(* Logix 5000 project; controller Battleship Emulate 5570 rev 32.11; software revision 32.00 *)

TASK MainTask (continuous, watchdog 500 ms) : MainProgram, Player_2, Player_1

MODULES
   Local : Emulate 5570 (ICP 2, rev 32.11)
END_MODULES

TYPE HMI_ScreenNames :
STRUCT
   LoadingScreen : STRING;
   BattleScreen : STRING;
END_STRUCT
END_TYPE

TYPE PlayerData :
STRUCT
   Ship : Ship[6];
   HMI : PlayerHMI;
   sName : STRING;
   nScore : INT;
   ShipSelectedFromFleet : SINT;
   sideShipSelected_ID : SINT;
   anySideShipSelected : BOOL;
   bShipsDeployed : BOOL;
   bTacticalScreenEnabled : BOOL;
   bBattleScreenEnabled : BOOL;
   bTurn : BOOL;
   bWinner : BOOL;
END_STRUCT
END_TYPE

TYPE PlayerHMI :
STRUCT
   sLoad_Or_Battle : STRING;   // The name of the screen that will load after player presses the Ready button
   bResetBoard_PB : BOOL;
   bRetrieveShip_PB : BOOL;
   bRetrieveShipPB_Vis : BOOL;
   bShipPiece_Orientation_PB : BOOL;
   bReady_PB : BOOL;   // Player Ready Signal from HMI
   bEnableStartPB : BOOL;   // Enable Start button on HMI
   bFight_PB : BOOL;
   bFightPB_Vis : BOOL;
   bWaitingForOpponent : BOOL;
END_STRUCT
END_TYPE

TYPE Ship :
STRUCT
   Position : INT[2];   // X-Y Ship Coordinates
   Pivot : INT[2];   // X-Y Pivot Coordinates
   nShipID : SINT;
   nShipLength : SINT;   // 5 = Carrier 4 = Battleship 3 = Cruiser 2 = Destroyer
   bIsHit : BOOL;
   bIsSunked : BOOL;
   bIsSelected : BOOL;
   bHideSidePiece : BOOL;
END_STRUCT
END_TYPE

TYPE Tile :
STRUCT
   IND : SINT;   // 0 = No ship 1 = Has ship 2 = Has ship and selected
   ShipID : SINT;
   hasShip : BOOL;
   squareSelected : BOOL;
END_STRUCT
END_TYPE

TYPE TileSelection :
STRUCT
   Coordinate : XYcoordinates;
   ShipId : DINT;
END_STRUCT
END_TYPE

TYPE top_scrn :
STRUCT
   notSelected : BOOL;
   selected : BOOL;
   hit : BOOL;
END_STRUCT
END_TYPE

TYPE XYcoordinates :
STRUCT
   row : SINT;
   column : SINT;
END_STRUCT
END_TYPE

ADD_ON_INSTRUCTION BattleTracker   (* revision 1.0 *)
VAR_IN_OUT
   TileSelected : TileSelection; {required}
   OtherPlayer_TS : Tile[11,11]; {required}
   BattleScreen : Tile[11,11]; {required}
   OtherPlayer : PlayerData; {required}
   ThisPlayer : PlayerData; {required}
END_VAR
VAR
   row : DINT; {access None}
   column : DINT; {access None}
END_VAR

ROUTINE Logic   (* structured text *)
   if OtherPlayer_TS[TileSelected.Coordinate.row, TileSelected.Coordinate.column].hasShip then
   	BattleScreen[TileSelected.Coordinate.row, TileSelected.Coordinate.column].IND := 4;
   	ThisPlayer.nScore := ThisPlayer.nScore + 1;
   else
   	BattleScreen[TileSelected.Coordinate.row, TileSelected.Coordinate.column].IND := 3;
   end_if;
   
   
   TileSelected.Coordinate.row := 0;
   TileSelected.Coordinate.column := 0;
   
   // Terminate player's turn
   ThisPlayer.bTurn := 0;
   OtherPlayer.bTurn := 1;
   
   
END_ROUTINE
END_ADD_ON_INSTRUCTION

ADD_ON_INSTRUCTION CommandShip   (* revision 1.0 *)
VAR_IN_OUT
   Player_Ship : Ship[5]; {required}
   Player_tacticalScreen : Tile[10,10]; {required}
END_VAR
VAR_INPUT
   verticalOrientation : BOOL; {required}
   NumberOfShips : DINT; {access Read Only, required}
END_VAR
VAR_IN_OUT
   shipSelected : SINT; {required}
END_VAR
VAR
   selectedSquare : XYcoordinates; {access None}
   x : DINT; {access None}
   row : DINT; {access None}
   column : DINT; {access None}
END_VAR

ROUTINE Logic   (* structured text *)
   // Initialize variables
   //shipSelected := -1;
   selectedSquare.row := -1;
   selectedSquare.column := -1;
   /*
   
   // Look for any side ship that was selected from the side pieces
   // shipSelected = the ship the was selected from the side pieces
   for x := 0 to NumberOfShips-1 by 1  do
   	//anySelected := 0;
   	if Player_Ship[x].isSelected then
   		shipSelected := x;
   		selectedSquare.row := -1;
   		selectedSquare.column := -1;
   	else
   		shipSelected := -1;
   		selectedSquare.row := -1;
   		selectedSquare.column := -1;
   	end_if;
   	/*
   	anySelected := ThisPlayer.Ship[x].isSelected OR anySelected;
   	if not anySelected then
   		shipSelected := -1;
   	end_if;
   
   
   end_for;
   
   */
   
   
   
   // If a ship piece was selected, enable search to look for the square that gets selected on the tactical screen
   // Store the XY coordinates of the selected square in selectedSquare.row and selectedSquare.column
   if shipSelected >= 0 then
   	for row := 0 to 9 by 1 do
   		for column := 0 to 9 by 1 do
   			if Player_tacticalScreen[row,column].squareSelected then
   				selectedSquare.row := row;
   				selectedSquare.column := column;
   				Player_tacticalScreen[row,column].squareSelected := 0;
   			end_if;
   		end_for;
   	end_for;
   end_if;
   
   
   /*
   // If a ship piece and a square were selected,
   // set the adjacent squares "hasShip" to 1 horizontally starting with the selected ship and moving to the right for as many squares as the ship's length
   if selectedSquare.row <> -1 AND selectedSquare.column <> -1 then
   
   	if verticalOrientation then		// Place ship in vertical orientation
   		for column := selectedSquare.column to selectedSquare.column + Player_Ship[x].shipLength -1 by 1 do
   			Player_tacticalScreen[selectedSquare.row,column].hasShip := 1;
   			Player_tacticalScreen[selectedSquare.row,column].hasShipType := shipSelected;
   			Player_tacticalScreen[selectedSquare.row,column].IND := 1;
   			Player_Ship[shipSelected].isSelected := 0;
   		end_for;
   
   
   	else	// Place ship in horizontal orientation
   		for row:= selectedSquare.row to selectedSquare.row + Player_Ship[x].shipLength -1 by 1 do
   			Player_tacticalScreen[row,selectedSquare.column].hasShip := 1;
   			Player_tacticalScreen[row,selectedSquare.column].hasShipType := shipSelected;
   			Player_tacticalScreen[row,selectedSquare.column].IND := 1;
   			Player_Ship[shipSelected].isSelected := 0;
   		end_for;
   	end_if;
   end_if;
   
   
   /*
   TODO
   
   add vertical/horizontal button and adjust how you lay the ship accordingly
   
   add retrieve button
   
   count down the ship pieces. disable piece once count reaches zero
   */
END_ROUTINE
END_ADD_ON_INSTRUCTION

ADD_ON_INSTRUCTION heartBeat   (* revision 1.0 *)
VAR_INPUT
   onTime : DINT; {required}
   offTime : DINT; {required}
END_VAR
VAR_OUTPUT
   Beat : BOOL; {access None, visible}
END_VAR
VAR
   T2 : TIMER; {access None}
   T1 : TIMER; {access None}
END_VAR

ROUTINE Logic   (* ladder *)
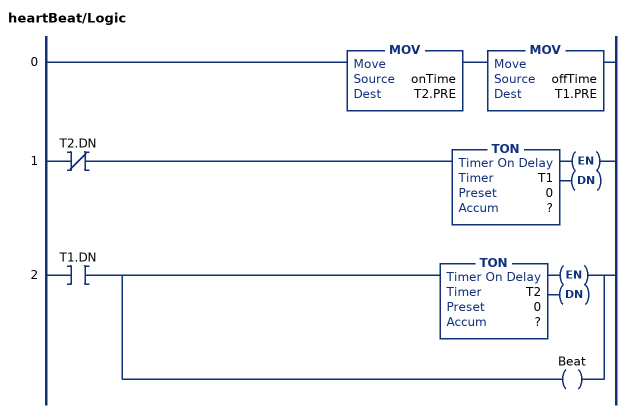
   0: MOV(onTime,T2.PRE)MOV(offTime,T1.PRE);
   1: XIO(T2.DN)TON(T1,?,?);
   2: XIC(T1.DN)[TON(T2,?,?) ,OTE(Beat) ];
END_ROUTINE
END_ADD_ON_INSTRUCTION

ADD_ON_INSTRUCTION InhibitTileSelect_BS   (* revision 1.0 *)
VAR_IN_OUT
   BattleScreen : Tile[11,11]; {required}
END_VAR
VAR
   row : DINT; {access None}
   column : DINT; {access None}
END_VAR

ROUTINE Logic   (* structured text *)
   for row := 1 to 10 by 1 do
   	for column := 1 to 10 by 1 do
   		BattleScreen [row, column].squareSelected := 0;
   	end_for;
   end_for;
END_ROUTINE
END_ADD_ON_INSTRUCTION

ADD_ON_INSTRUCTION PlaceShip   (* revision 1.0 *)
VAR_IN_OUT
   Player : PlayerData; {required}
   SelectedTile : TileSelection; {required}
   TacticalScreen : Tile[11,11]; {required}
END_VAR
VAR_INPUT
   PlaceShipReq : BOOL; {access Read Only, required}
END_VAR
VAR_OUTPUT
   bShipCollision : BOOL; {access None, visible}
   bShipOutOfBounds : BOOL; {access None, visible}
END_VAR
VAR
   row : DINT; {access None}
   column : DINT; {access None}
END_VAR

ROUTINE Logic   (* structured text *)
   // Initialize variables when the AOI is called
   if PlaceShipReq then
   	bShipCollision := 0;
   	bShipOutOfBounds := 0;
   end_if;
   
   
   // Detrmine ship orientation (horizontal or vertical)
   if Player.HMI.bShipPiece_Orientation_PB then
   //---------------------------------------------------------------------------------------------
   //									Vertical placement
   //---------------------------------------------------------------------------------------------
   
   	// Check if the ship can be placed on the board (out of bounds check)
   	// Raise a flag and display a warning if the user tried to place a ship out of bounds (see Messages routine)
   	if SelectedTile.Coordinate.row + Player.Ship[Player.sideShipSelected_ID].nShipLength > 11 then
   		bShipOutOfBounds := 1;
   	end_if;
   
   
   	// Check if there is no collision with other ships
   	// Raise a flag and display a warning if the user tried to place a ship on top of another (see Messages routine)
   	if not bShipOutOfBounds then
   		for row := SelectedTile.Coordinate.row to SelectedTile.Coordinate.row + Player.Ship[Player.sideShipSelected_ID].nShipLength -1 by 1 do
   			if TacticalScreen[row,SelectedTile.Coordinate.column].hasShip then
   				bShipCollision := 1;
   			end_if;
   		end_for;
   	end_if;
   
   
   	// Place ship if not out of bounds and no collision
   	if not (bShipCollision or bShipOutOfBounds) then
   		// Move vertically across rows
   		for row := SelectedTile.Coordinate.row to SelectedTile.Coordinate.row + Player.Ship[Player.sideShipSelected_ID].nShipLength -1 by 1 do
   
   			// Set tile ship status (has ship)
   			TacticalScreen[row,SelectedTile.Coordinate.column].hasShip := 1;
   			// Set ID of the ship in that tile
   			TacticalScreen[row,SelectedTile.Coordinate.column].ShipID :=Player.sideShipSelected_ID;
   			// Set tile indicator (change tile color in the HMI)
   			TacticalScreen[row,SelectedTile.Coordinate.column].IND := 1;
   		end_for;
   
   		// Hide ship token
   		Player.Ship[Player.sideShipSelected_ID].bHideSidePiece := 1;
   	end_if;
   
   
   else
   //---------------------------------------------------------------------------------------------
   //									Horizontal placement
   //---------------------------------------------------------------------------------------------
   
   
   	// Check if the ship can be placed on the board (out of bounds check)
   	// Raise a flag and display a warning if the user tried to place a ship out of bounds (see Messages routine)
   	if SelectedTile.Coordinate.column + Player.Ship[Player.sideShipSelected_ID].nShipLength > 11 then
   		bShipOutOfBounds := 1;
   	end_if;
   
   
   	// Check if there is no collision with other ships
   	// Raise a flag and display a warning if the user tried to place a ship on top of another (see Messages routine)
   	if not bShipOutOfBounds then
   		for column := SelectedTile.Coordinate.column to SelectedTile.Coordinate.column + Player.Ship[Player.sideShipSelected_ID].nShipLength -1 by 1 do
   			if TacticalScreen[SelectedTile.Coordinate.row,column].hasShip then
   				bShipCollision := 1;
   			end_if;
   		end_for;
   	end_if;
   
   
   
   	// Place ship if not out of bounds and no collision
   	if not (bShipCollision or bShipOutOfBounds) then
   		// Move horizontally across columns
   		for column := SelectedTile.Coordinate.column to SelectedTile.Coordinate.column + Player.Ship[Player.sideShipSelected_ID].nShipLength -1 by 1 do
   
   			// Set tile ship status (has ship)
   			TacticalScreen[SelectedTile.Coordinate.row,column].hasShip := 1;
   			// Set ID of the ship in that tile
   			TacticalScreen[SelectedTile.Coordinate.row,column].ShipID := Player.sideShipSelected_ID;
   			// Set tile indicator (change tile color in the HMI)
   			TacticalScreen[SelectedTile.Coordinate.row,column].IND := 1;
   		end_for;
   
   		// Hide ship token
   		Player.Ship[Player.sideShipSelected_ID].bHideSidePiece := 1;
   	end_if;
   end_if;
   
   
   // Clear selected tile X-Y coordinates
   // This is necesary because if a ship is placed and the selected tile coordinates are not cleared, the AOI will try to place another ship when the user selects one of the token ships
   SelectedTile.Coordinate.row := 0;
   SelectedTile.Coordinate.column := 0;
   
   // Clear token ID from memory
   Player.sideShipSelected_ID := 0;
END_ROUTINE
END_ADD_ON_INSTRUCTION

ADD_ON_INSTRUCTION ResetTacticalScreen   (* revision 1.0 *)
VAR_IN_OUT
   NULL_TaclticalScreen : Tile; {required}
   TacticalScreen : Tile[11,11]; {required}
   BattleScreen : Tile[11,11]; {required}
END_VAR
VAR
   row : SINT; {access None}
   column : SINT; {access None}
END_VAR

ROUTINE Logic   (* structured text *)
   for row := 0 to 10 by 1 do
   	for column := 0 to 10 by 1 do
   
   		// Reset Tactical Screen
   		TacticalScreen[row,column].hasShip := NULL_TaclticalScreen.hasShip;
   		TacticalScreen[row,column].ShipID := NULL_TaclticalScreen.ShipID;
   		TacticalScreen[row,column].IND := NULL_TaclticalScreen.IND;
   		TacticalScreen[row,column].squareSelected := NULL_TaclticalScreen.squareSelected;
   
   		// Reset Battle Screen
   		BattleScreen[row,column].IND := 0;
   	end_for;
   end_for;
END_ROUTINE
END_ADD_ON_INSTRUCTION

ADD_ON_INSTRUCTION RetrieveShip   (* revision 1.0 *)
VAR_IN_OUT
   Tile : TileSelection; {required}
   TacticalScreen : Tile[11,11]; {required}
   Player : PlayerData; {required}
END_VAR
VAR
   row : DINT; {access None}
   column : DINT; {access None}
END_VAR

ROUTINE Logic   (* structured text *)
   
   
   for row := 1 to 10 by 1 do
   	for column := 1 to 10 by 1 do
   		if TacticalScreen [row, column].ShipID = Tile.ShipId then
   			TacticalScreen [row, column].ShipID := 0;
   			TacticalScreen [row, column].hasShip := 0;
   			TacticalScreen [row, column].IND := 0;
   		end_if;
   	end_for;
   end_for;
   
   Player.Ship[Tile.ShipId].bHideSidePiece := 0;
   
   
   
   
   
   
   
   
   
   
   
   
   
   
   
   
   
   
   
   
   /*
   //Initialize variables
   if not squareSelected then
   	row := -1;
   	column := -1;
   end_if;
   
   
   for row := 0 to 9 by 1 do
   	for column := 0 to 9 by 1 do
   		if Player_tacticalScreen[row,column].squareSelected AND Player_tacticalScreen[row,column].hasShip then
   			selectedSquare.row := row;
   			selectedSquare.column := column;
   			selectedShipType := Player_tacticalScreen[row,column].ShipID;
   			squareSelected := 1;
   			Player_tacticalScreen[row,column].squareSelected := 0;
   		end_if;
   		/*
   		if P1_tacticalScreen[row,column].squareSelected AND P1_tacticalScreen[row,column].IND = 2 then
   			squareSelected := 0;
   			P1_tacticalScreen[row,column].IND := 1;
   		end_if;
   		*/
   /*
   	end_for;
   end_for;
   
   
   if squareSelected then
   	for row := 0 to 9 by 1 do
   		for column := 0 to 9 by 1 do
   			if Player_tacticalScreen[row,column].ShipID = selectedShipType then;
   				Player_tacticalScreen[row,column].IND := 2;
   				readyToRetrieve := 1;
   				squareSelected := 0;
   			end_if;
   		end_for;
   	end_for;
   end_if;
   
   if readyToRetrieve AND RetrieveShip then
   	for row := 0 to 9 by 1 do
   		for column := 0 to 9 by 1 do
   			if Player_tacticalScreen[row,column].ShipID = selectedShipType then;
   				Player_tacticalScreen[row,column].hasShip := 0;
   				Player_tacticalScreen[row,column].IND := 0;
   				Player_tacticalScreen[row,column].ShipID := -1;
   				readyToRetrieve := 0;
   				squareSelected := 0;
   			end_if;
   		end_for;
   	end_for;
   end_if;
   
   
   if squareSelected AND Player_tacticalScreen[selectedSquare.row,selectedSquare.column].IND = 2 then
   	for row := 0 to 9 by 1 do
   		for column := 0 to 9 by 1 do
   			if Player_tacticalScreen[row,column].ShipID = selectedShipType then;
   				Player_tacticalScreen[row,column].IND := 1;
   				readyToRetrieve := 0;
   				squareSelected := 0;
   			end_if;
   		end_for;
   	end_for;
   end_if;
   */
END_ROUTINE
END_ADD_ON_INSTRUCTION

ADD_ON_INSTRUCTION SideShips   (* revision 1.0 *)
VAR_IN_OUT
   Player_Ship : Ship[5]; {required}
END_VAR
VAR_OUTPUT
   shipSelected : SINT; {required}
END_VAR
VAR
   shipCount : SINT; {access None}
   shipSelected_OSR : FBD_ONESHOT[9]; {access None}
   aShipWasSelected : BOOL[32]; {access None}
END_VAR

ROUTINE Logic   (* structured text *)
   // This code handles the ship pieces tha get selected on the left of the tactical screen
   
   // Look for a one shot rising that comes from pressing on one ship piece. Save which ship piece was selected to shipSelected
   
   
   for shipCount:=0 to 8 by 1 do
   	if not Player_Ship[shipCount].bIsSelected then
   		shipSelected := -1;
   	end_if;
   
   	shipSelected_OSR[shipCount].InputBit := Player_Ship[shipCount].bIsSelected;
   	OSRI(shipSelected_OSR[shipCount]);
   	aShipWasSelected[shipCount] := shipSelected_OSR[shipCount].OutputBit;
   
   	if aShipWasSelected[shipCount] then
   		shipSelected := shipCount;
   	end_if;
   end_for;
   
   
   if aShipWasSelected[0] or aShipWasSelected[1] or aShipWasSelected[2] or aShipWasSelected[3] or aShipWasSelected[4] or aShipWasSelected[5] then
   	aShipWasSelected[10] := 1;
   end_if;
   
   if aShipWasSelected[6] or aShipWasSelected[7] or aShipWasSelected[8] or aShipWasSelected[9] then
   	aShipWasSelected[11] := 1;
   end_if;
   
   // If ANY ship was selected then NONE of the other ships can be selected, set isSelected (for the rest of the ships) to zero
   if aShipWasSelected[10] or aShipWasSelected[11] then
   	for shipCount:=0 to 8 by 1 do
   		if shipCount <> shipSelected then
   			Player_Ship[shipCount].bIsSelected := 0;
   		end_if;
   	end_for;
   end_if;
   
   /*
   TODO
   
   Keep count of how many ship pieces are left
   */
END_ROUTINE
END_ADD_ON_INSTRUCTION

ADD_ON_INSTRUCTION TileDetection   (* revision 1.0 *)
VAR_IN_OUT
   Screen : Tile[11,11]; {required}
   SelectedTile : TileSelection; {required}
   Player : PlayerData; {required}
END_VAR
VAR_INPUT
   bShipCollision : BOOL; {access Read Only, required}
END_VAR
VAR
   row : DINT; {access None}
   column : DINT; {access None}
   bSomeShipSelected : BOOL; {access None}
   nSelectedTile_ShipIDEcho : DINT; {access None}
END_VAR

ROUTINE Logic   (* structured text *)
   /*
   -------------------------------------------------------------------------------------------------
   	This FB Scans the Tactical Screen and returns the X-Y coordinates of the tile that was selected
   	It also returns the ShipID of the ship placed in the selected tile
   
   
   -------------------------------------------------------------------------------------------------
   */
   
   bSomeShipSelected := 0;
   
   
   // Scan the Tactical Screen to see which tile was selected
   // Store the X-Y coordinates and ship ID (if any). Set the button back to an open state
   for row := 1 to 10 by 1 do
   	for column := 1 to 10 by 1 do
   		if Screen[row,column].squareSelected then
   
   			SelectedTile.Coordinate.row := row;
   			SelectedTile.Coordinate.column := column;
   			SelectedTile.ShipId := Screen[row,column].ShipID;
   			// nSelectedTile_ShipIDEcho := TacticalScreen[row,column].ShipID;
   
   
   
   
   
   
   			Screen[row,column].squareSelected := 0;
   		end_if;
   	end_for;
   end_for;
   
   
   
   for row := 1 to 10 by 1 do
   	for column := 1 to 10 by 1 do
   		if Screen[row,column].IND = 2 then
   			bSomeShipSelected := 1;
   		end_if;
   	end_for;
   end_for;
   
   
   
   
   
   
   
   
   for row := 1 to 10 by 1 do
   	for column := 1 to 10 by 1 do
   		if Screen[row,column].ShipID = SelectedTile.ShipId and SelectedTile.ShipId > 0 and Player.sideShipSelected_ID = 0 and not bShipCollision and not bSomeShipSelected and Screen[row,column].IND <> 2 then
   			Screen[row,column].IND := 2;
   			// nSelectedTile_ShipIDEcho := 0;
   		end_if;
   	end_for;
   end_for;
   
   
   /*
   
   for row := 1 to 10 by 1 do
   	for column := 1 to 10 by 1 do
   		if TacticalScreen[row,column].ShipID = nSelectedTile_ShipIDEcho and TacticalScreen[row,column].IND = 2 then
   			TacticalScreen[row,column].IND := 1;
   		end_if;
   	end_for;
   end_for;
   */
   
   
   // Clear the X-Y coordinates of the selected tile in the Tactical Screen if no token was selected and the tile selected is empty (has no ship)
   if Player.bTacticalScreenEnabled and Player.sideShipSelected_ID = 0 and NOT Screen[SelectedTile.Coordinate.row, SelectedTile.Coordinate.column].hasShip then
   	SelectedTile.Coordinate.row := 0;
   	SelectedTile.Coordinate.column := 0;
   end_if;
END_ROUTINE
END_ADD_ON_INSTRUCTION

VAR_GLOBAL   (* controller tags *)
   anySelected : BOOL;
   bDebbugOn : BOOL := 1;
   column : DINT := 11;
   HeartBeat : BOOL := 1;
   HMI_Macro_ResetBoard : BOOL; {access Read Only}
   Macro_ResetBoard : BOOL; {access Read Only}
   nMaximunScore : DINT := 17; {constant, access Read Only}
   NULL_PlayerHMI : PlayerHMI; {constant, access Read Only}
   NULL_Ship : Ship; {constant, access Read Only}
   NULL_TaclticalScreen : Tile; {access Read Only}
   NULL_TileSelection : TileSelection; {constant, access Read Only}
   NumberOfShips : SINT := 5;
   P1_BattleScreen : Tile[11,11];
   P1_tacticalScreen : Tile[11,11];
   P2_tacticalScreen : Tile[11,11];
   pHMI_Macro_ResetBoard_ONS : BOOL; {access Read Only}
   Player1 : PlayerData := (Ship[1].nShipID := 1, Ship[1].nShipLength := 5, Ship[2].nShipID := 2, Ship[2].nShipLength := 4, Ship[3].nShipID := 3, Ship[3].nShipLength := 3, Ship[4].nShipID := 4, Ship[4].nShipLength := 3, Ship[5].nShipID := 5, Ship[5].nShipLength := 2, HMI.sLoad_Or_Battle := '1_BattleScreen', HMI.bReady_PB := 1, HMI.bEnableStartPB := 1, sName := 'Jeyc', bTacticalScreenEnabled := 1);
   Player2 : PlayerData := (HMI.bReady_PB := 1, sName := 'Player 2');
   row : DINT := 11;
   ScreenNamesData : HMI_ScreenNames := (LoadingScreen := '0_LoadingScreen', BattleScreen := '1_BattleScreen'); {constant, access Read Only}
   selectedSquare : XYcoordinates := (row := -1, column := -1);
   SelectedTileShipID : SINT;
END_VAR

PROGRAM MainProgram   (* main routine MainRoutine *)
VAR
   EQU_01 : FBD_COMPARE := (SourceB := 17.0);
   EQU_02 : FBD_COMPARE := (SourceB := 17.0);
   Heart : heartBeat := (onTime := 500, offTime := 500, Beat := 1);
END_VAR

ROUTINE MainRoutine   (* ladder *)
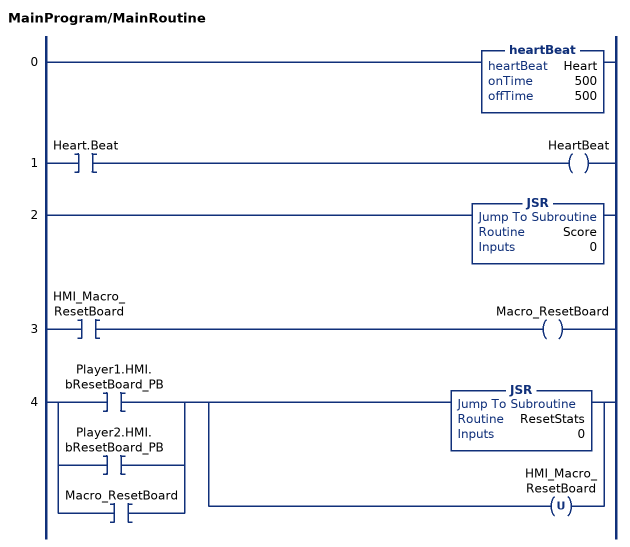
   0: heartBeat(Heart,500,500);
   1: XIC(Heart.Beat)OTE(HeartBeat);
   2: JSR(Score,0);
   3: XIC(HMI_Macro_ResetBoard)OTE(Macro_ResetBoard);
   4: [XIC(Player1.HMI.bResetBoard_PB) ,XIC(Player2.HMI.bResetBoard_PB) ,XIC(Macro_ResetBoard) ][JSR(ResetStats,0) ,OTU(HMI_Macro_ResetBoard) ];
END_ROUTINE

ROUTINE ResetStats   (* ladder *)
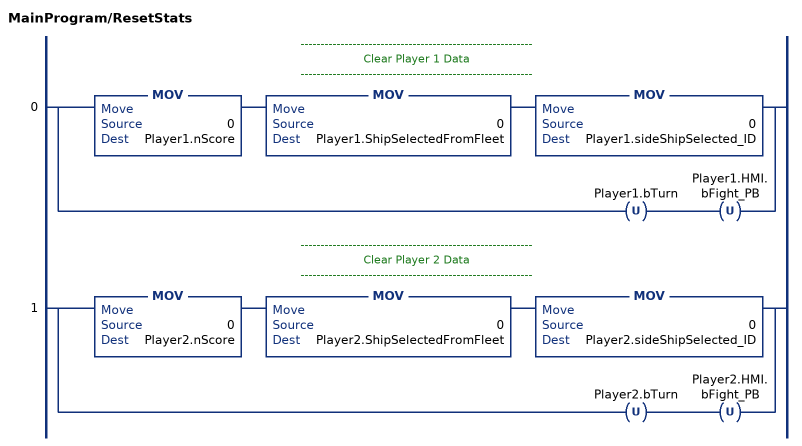
   // ----------------------------------------------------------
   // Clear Player 1 Data
   // ----------------------------------------------------------
   0: [MOV(0,Player1.nScore) MOV(0,Player1.ShipSelectedFromFleet) MOV(0,Player1.sideShipSelected_ID) ,OTU(Player1.bTurn) OTU(Player1.HMI.bFight_PB) ];
   // ----------------------------------------------------------
   // Clear Player 2 Data
   // ----------------------------------------------------------
   1: [MOV(0,Player2.nScore) MOV(0,Player2.ShipSelectedFromFleet) MOV(0,Player2.sideShipSelected_ID) ,OTU(Player2.bTurn) OTU(Player2.HMI.bFight_PB) ];
END_ROUTINE

ROUTINE Score   (* function block diagram *)
   SHEET 1
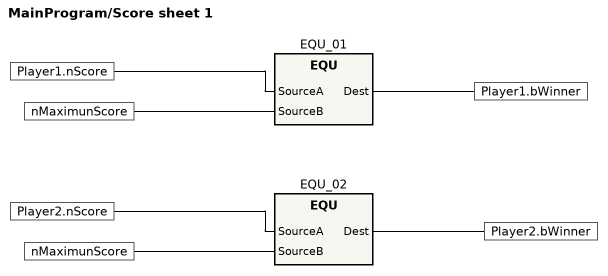
   EQU_01 : EQU(SourceA := Player1.nScore, SourceB := nMaximunScore);
   EQU_02 : EQU(SourceA := Player2.nScore, SourceB := nMaximunScore);
   Player1.bWinner := EQU_01.Dest;
   Player2.bWinner := EQU_02.Dest;
END_ROUTINE
END_PROGRAM

PROGRAM Player_1   (* main routine Main *)
VAR
   AOI_BattleTracker : BattleTracker;
   AOI_BSTileDetection : TileDetection;
   AOI_InhbTileSelec : InhibitTileSelect_BS;
   AOI_PlaceShip : PlaceShip;
   AOI_ResetScreen : ResetTacticalScreen;
   AOI_RetrieveShip : RetrieveShip;
   AOI_TSTileDetection : TileDetection;
   BattleScreen_SelectedTile : TileSelection;
   cntr : SINT := 6;
   CurrentMessages : DINT[10];
   CycleLoadingTime : DINT := 5000;
   dosomething : BOOL;
   DotOff : SINT := 2;
   DotOff_Time : REAL[9] := ([0] := 625.0, [1] := 1250.0, [2] := 1875.0, [3] := 2500.0, [4] := 3125.0, [5] := 3750.0, [6] := 4375.0, [7] := 5000.0);
   LoadingDots : TIMER := (PRE := 5000, ACC := 906, EN := 1, TT := 1);
        .PRE   // Use this to change how fast the loading dots move
   Message_TMR : TIMER[20] := ([0].PRE := 5000, [1].PRE := 5000);
   MessageCmpControl : CONTROL := (LEN := 320, IN := 1);
   MessageReference : DINT[10];
   MessageResultControl : CONTROL := (LEN := 1);
   MessageResults : DINT[1];
   Messages : DINT;
   MessageScrollTimer : TIMER := (PRE := 2000);
   OtherPlayer : ALIAS FOR Player2;
   pMessage1_ONS : BOOL := 1;
   pPlaceShip_ONS : BOOL;
   pResetBoard_ONS : BOOL;
   RetrieveShips : RetrieveShip;   // Handles ship retrieving process
   rtrv_column : DINT := 10;
   rtrv_column2 : DINT;
   rtrv_row : DINT := 10;
   rtrv_row2 : DINT;
   rtv_selectedSquare : XYcoordinates;
   shipSelected_OSR : FBD_ONESHOT[15];
   StartFight_TMR : TIMER := (PRE := 1000); {access Read Only}
   TacticalScreen_SelectedTile : TileSelection;
   ThisPlayer : ALIAS FOR Player1;
        .Ship[0]   // Null Ship
END_VAR

ROUTINE HMI   (* ladder *)
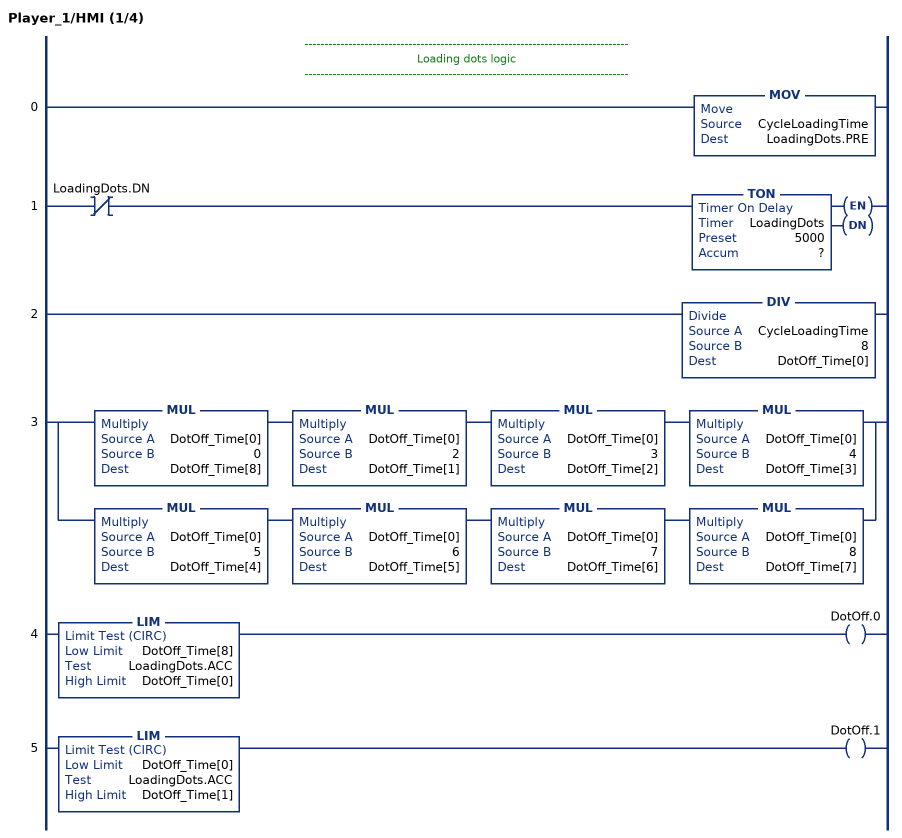
   // ---------------------------------------------------------------------------------
   // Loading dots logic
   // ---------------------------------------------------------------------------------
   0: MOV(CycleLoadingTime,LoadingDots.PRE);
   1: XIO(LoadingDots.DN)TON(LoadingDots,?,?);
   2: DIV(CycleLoadingTime,8,DotOff_Time[0]);
   3: [MUL(DotOff_Time[0],0,DotOff_Time[8]) MUL(DotOff_Time[0],2,DotOff_Time[1]) MUL(DotOff_Time[0],3,DotOff_Time[2]) MUL(DotOff_Time[0],4,DotOff_Time[3]) ,MUL(DotOff_Time[0],5,DotOff_Time[4]) MUL(DotOff_Time[0],6,DotOff_Time[5]) MUL(DotOff_Time[0],7,DotOff_Time[6]) MUL(DotOff_Time[0],8,DotOff_Time[7]) ];
   4: LIM(DotOff_Time[8],LoadingDots.ACC,DotOff_Time[0])OTE(DotOff.0);
   5: LIM(DotOff_Time[0],LoadingDots.ACC,DotOff_Time[1])OTE(DotOff.1);
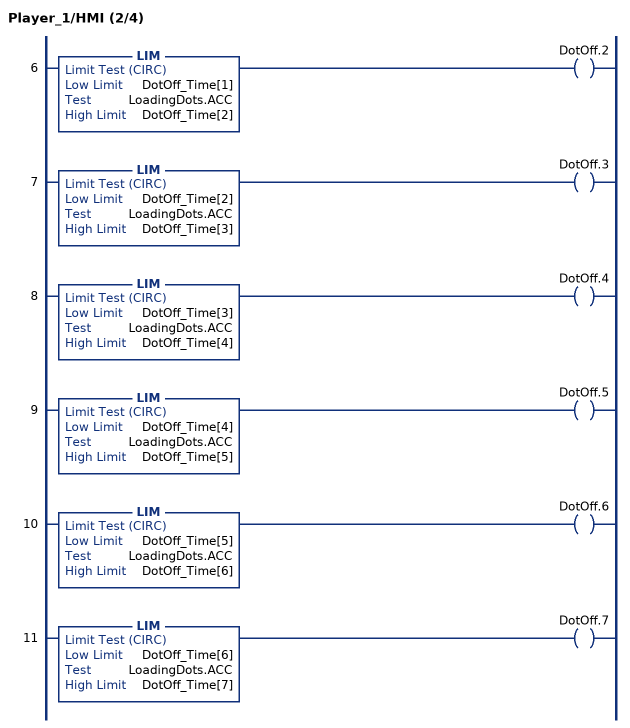
   6: LIM(DotOff_Time[1],LoadingDots.ACC,DotOff_Time[2])OTE(DotOff.2);
   7: LIM(DotOff_Time[2],LoadingDots.ACC,DotOff_Time[3])OTE(DotOff.3);
   8: LIM(DotOff_Time[3],LoadingDots.ACC,DotOff_Time[4])OTE(DotOff.4);
   9: LIM(DotOff_Time[4],LoadingDots.ACC,DotOff_Time[5])OTE(DotOff.5);
   10: LIM(DotOff_Time[5],LoadingDots.ACC,DotOff_Time[6])OTE(DotOff.6);
   11: LIM(DotOff_Time[6],LoadingDots.ACC,DotOff_Time[7])OTE(DotOff.7);
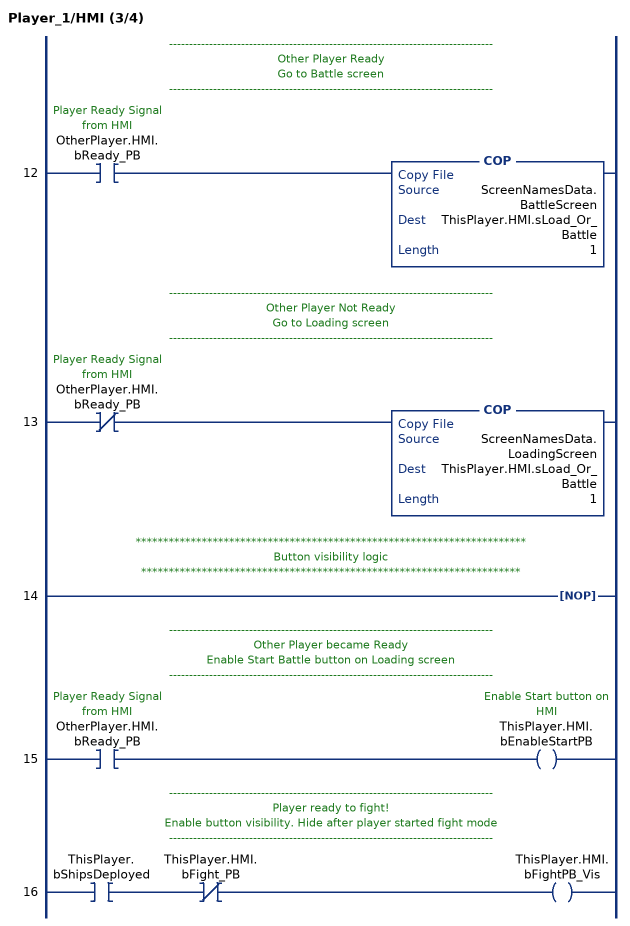
   // ---------------------------------------------------------------------------------
   // Other Player Ready
   // Go to Battle screen
   // ---------------------------------------------------------------------------------
   12: XIC(OtherPlayer.HMI.bReady_PB)COP(ScreenNamesData.BattleScreen,ThisPlayer.HMI.sLoad_Or_Battle,1);
   // ---------------------------------------------------------------------------------
   // Other Player Not Ready
   // Go to Loading screen
   // ---------------------------------------------------------------------------------
   13: XIO(OtherPlayer.HMI.bReady_PB)COP(ScreenNamesData.LoadingScreen,ThisPlayer.HMI.sLoad_Or_Battle,1);
   // ***********************************************************************
   // Button visibility logic
   // *********************************************************************
   14: NOP();
   // ---------------------------------------------------------------------------------
   // Other Player became Ready
   // Enable Start Battle button on Loading screen
   // ---------------------------------------------------------------------------------
   15: XIC(OtherPlayer.HMI.bReady_PB)OTE(ThisPlayer.HMI.bEnableStartPB);
   // ---------------------------------------------------------------------------------
   // Player ready to fight!
   // Enable button visibility. Hide after player started fight mode
   // ---------------------------------------------------------------------------------
   16: XIC(ThisPlayer.bShipsDeployed)XIO(ThisPlayer.HMI.bFight_PB)OTE(ThisPlayer.HMI.bFightPB_Vis);
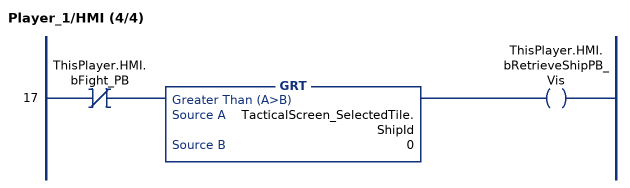
   17: XIO(ThisPlayer.HMI.bFight_PB)GRT(TacticalScreen_SelectedTile.ShipId,0)OTE(ThisPlayer.HMI.bRetrieveShipPB_Vis);
END_ROUTINE

ROUTINE Main   (* ladder *)
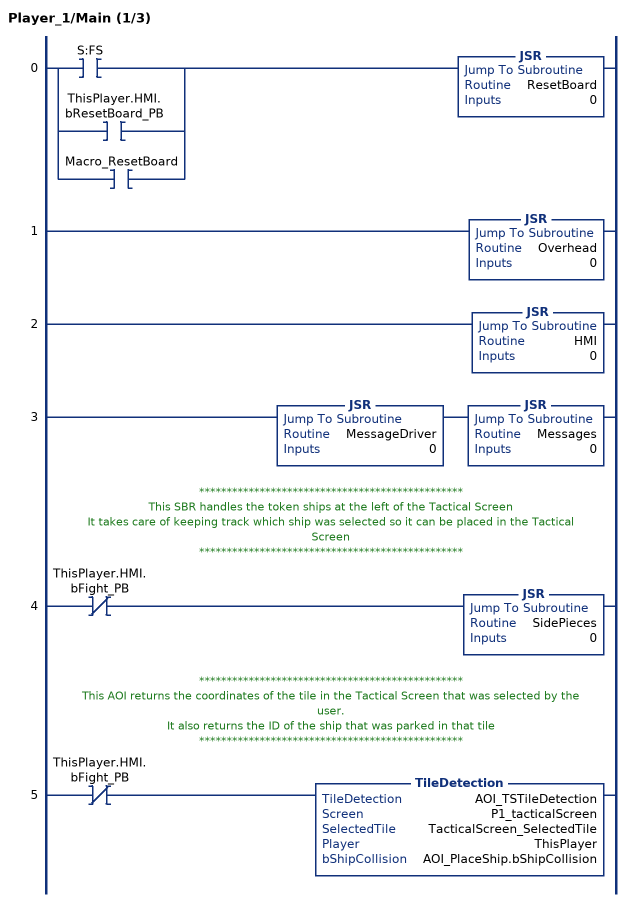
   0: [XIC(S:FS) ,XIC(ThisPlayer.HMI.bResetBoard_PB) ,XIC(Macro_ResetBoard) ]JSR(ResetBoard,0);
   1: JSR(Overhead,0);
   2: JSR(HMI,0);
   3: JSR(MessageDriver,0)JSR(Messages,0);
   // ************************************************
   // This SBR handles the token ships at the left of the Tactical Screen
   // It takes care of keeping track which ship was selected so it can be placed in the Tactical Screen
   // ************************************************
   4: XIO(ThisPlayer.HMI.bFight_PB)JSR(SidePieces,0);
   // ************************************************
   // This AOI returns the coordinates of the tile in the Tactical Screen that was selected by the user.
   // It also returns the ID of the ship that was parked in that tile
   // ************************************************
   5: XIO(ThisPlayer.HMI.bFight_PB)TileDetection(AOI_TSTileDetection,P1_tacticalScreen,TacticalScreen_SelectedTile,ThisPlayer,AOI_PlaceShip.bShipCollision);
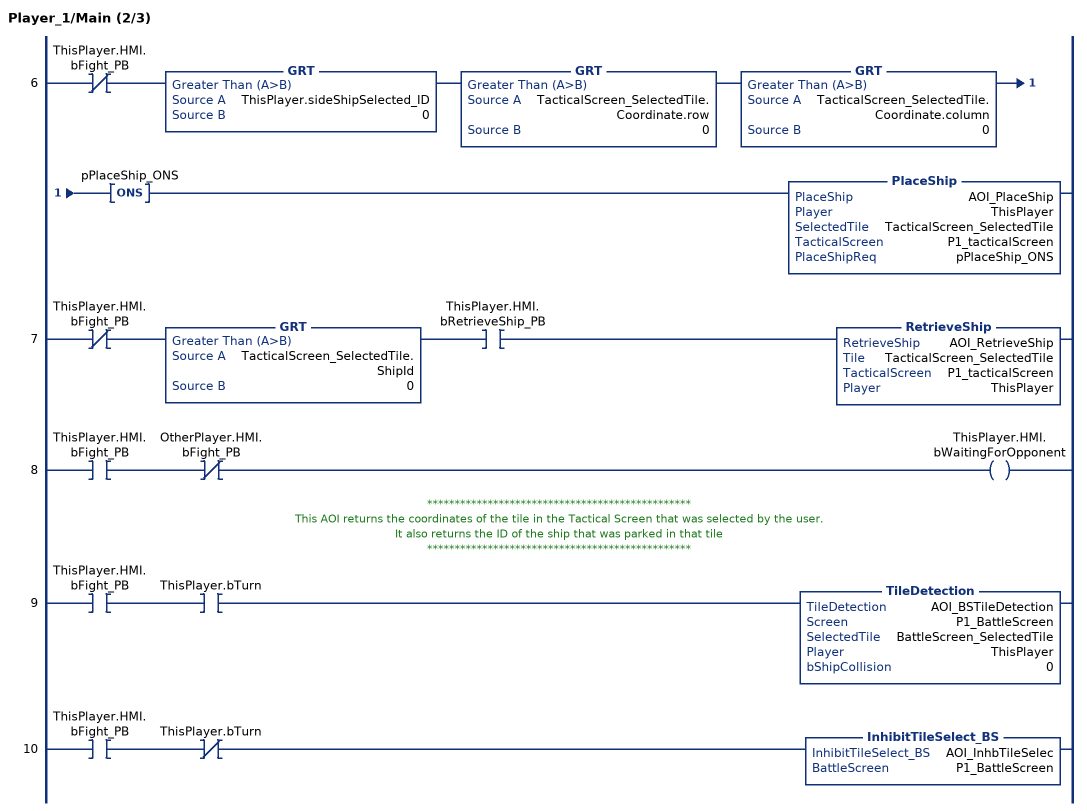
   6: XIO(ThisPlayer.HMI.bFight_PB)GRT(ThisPlayer.sideShipSelected_ID,0)GRT(TacticalScreen_SelectedTile.Coordinate.row,0)GRT(TacticalScreen_SelectedTile.Coordinate.column,0)ONS(pPlaceShip_ONS)PlaceShip(AOI_PlaceShip,ThisPlayer,TacticalScreen_SelectedTile,P1_tacticalScreen,pPlaceShip_ONS);
   7: XIO(ThisPlayer.HMI.bFight_PB)GRT(TacticalScreen_SelectedTile.ShipId,0)XIC(ThisPlayer.HMI.bRetrieveShip_PB)RetrieveShip(AOI_RetrieveShip,TacticalScreen_SelectedTile,P1_tacticalScreen,ThisPlayer);
   8: XIC(ThisPlayer.HMI.bFight_PB)XIO(OtherPlayer.HMI.bFight_PB)OTE(ThisPlayer.HMI.bWaitingForOpponent);
   // ************************************************
   // This AOI returns the coordinates of the tile in the Tactical Screen that was selected by the user.
   // It also returns the ID of the ship that was parked in that tile
   // ************************************************
   9: XIC(ThisPlayer.HMI.bFight_PB)XIC(ThisPlayer.bTurn)TileDetection(AOI_BSTileDetection,P1_BattleScreen,BattleScreen_SelectedTile,ThisPlayer,0);
   10: XIC(ThisPlayer.HMI.bFight_PB)XIO(ThisPlayer.bTurn)InhibitTileSelect_BS(AOI_InhbTileSelec,P1_BattleScreen);
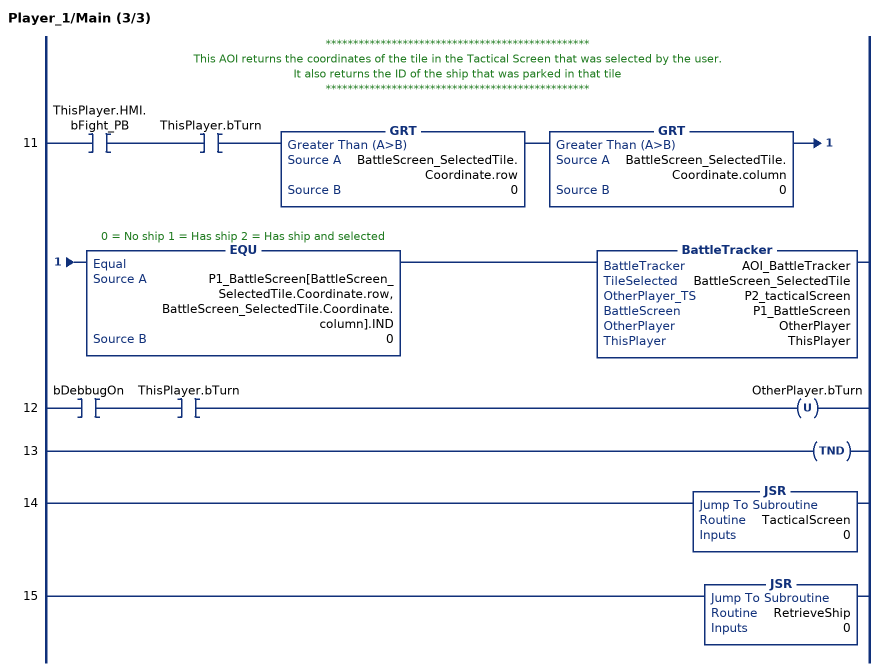
   // ************************************************
   // This AOI returns the coordinates of the tile in the Tactical Screen that was selected by the user.
   // It also returns the ID of the ship that was parked in that tile
   // ************************************************
   11: XIC(ThisPlayer.HMI.bFight_PB)XIC(ThisPlayer.bTurn)GRT(BattleScreen_SelectedTile.Coordinate.row,0)GRT(BattleScreen_SelectedTile.Coordinate.column,0)EQU(P1_BattleScreen[BattleScreen_SelectedTile.Coordinate.row, BattleScreen_SelectedTile.Coordinate.column].IND,0)BattleTracker(AOI_BattleTracker,BattleScreen_SelectedTile,P2_tacticalScreen,P1_BattleScreen,OtherPlayer,ThisPlayer);
   12: XIC(bDebbugOn)XIC(ThisPlayer.bTurn)OTU(OtherPlayer.bTurn);
   13: TND();
   14: JSR(TacticalScreen,0);
   15: JSR(RetrieveShip,0);
END_ROUTINE

ROUTINE MessageDriver   (* ladder *)
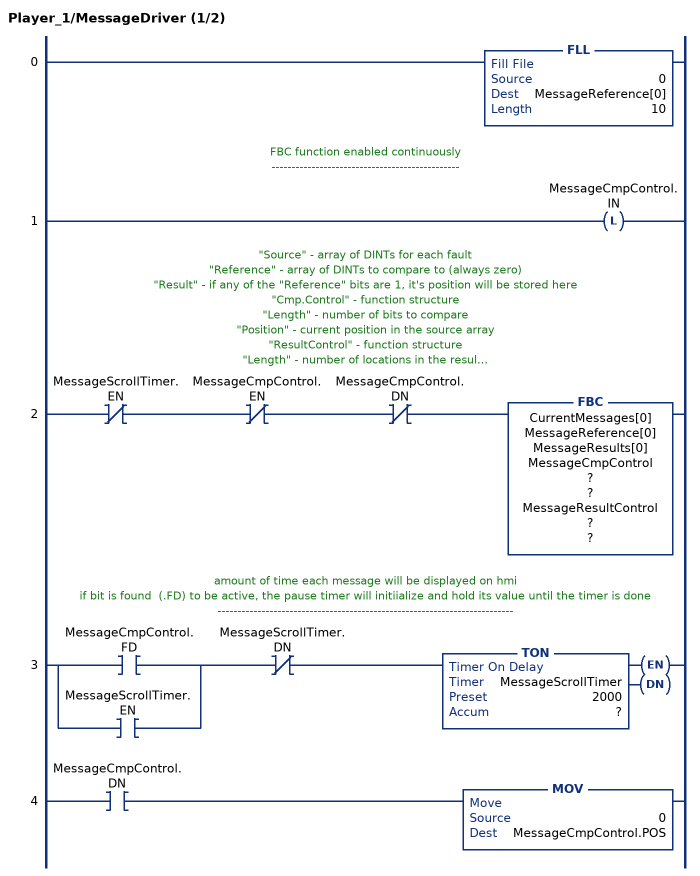
   0: FLL(0,MessageReference[0],10);
   // FBC function enabled continuously
   // -----------------------------------------------
   1: OTL(MessageCmpControl.IN);
   // "Source" - array of DINTs for each fault
   // "Reference" - array of DINTs to compare to (always zero)
   // "Result" - if any of the "Reference" bits are 1, it's position will be stored here
   // "Cmp.Control" - function structure
   // "Length" - number of bits to compare
   // "Position" - current position in the source array
   // "ResultControl" - function structure
   // "Length" - number of locations in the result
   // "Position" - current position in result
   // ------------------------------------------------------------------------
   // as long as the display timer is not running, this function will scroll continuously looking for a bit to be active (1)
   2: XIO(MessageScrollTimer.EN)XIO(MessageCmpControl.EN)XIO(MessageCmpControl.DN)FBC(CurrentMessages[0],MessageReference[0],MessageResults[0],MessageCmpControl,?,?,MessageResultControl,?,?);
   // amount of time each message will be displayed on hmi
   // if bit is found  (.FD) to be active, the pause timer will initiialize and hold its value until the timer is done
   // --------------------------------------------------------------------------
   3: [XIC(MessageCmpControl.FD) ,XIC(MessageScrollTimer.EN) ]XIO(MessageScrollTimer.DN)TON(MessageScrollTimer,?,?);
   4: XIC(MessageCmpControl.DN)MOV(0,MessageCmpControl.POS);
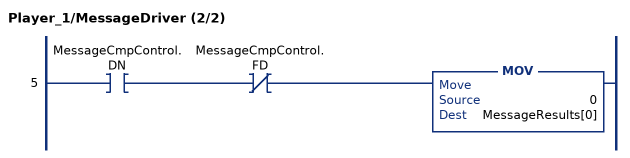
   5: XIC(MessageCmpControl.DN)XIO(MessageCmpControl.FD)MOV(0,MessageResults[0]);
END_ROUTINE

ROUTINE Messages   (* ladder *)
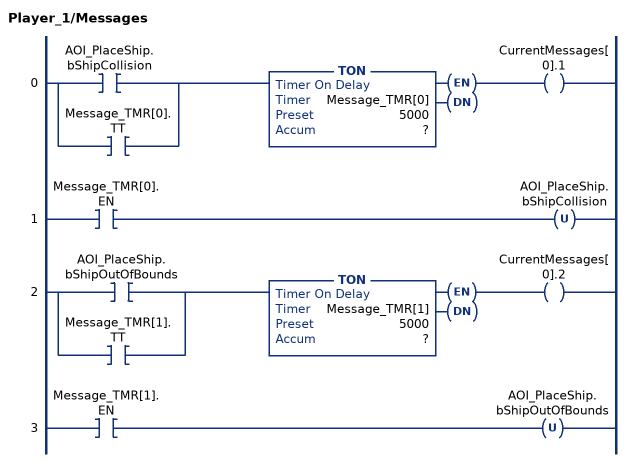
   0: [XIC(AOI_PlaceShip.bShipCollision) ,XIC(Message_TMR[0].TT) ]TON(Message_TMR[0],?,?)OTE(CurrentMessages[0].1);
   1: XIC(Message_TMR[0].EN)OTU(AOI_PlaceShip.bShipCollision);
   2: [XIC(AOI_PlaceShip.bShipOutOfBounds) ,XIC(Message_TMR[1].TT) ]TON(Message_TMR[1],?,?)OTE(CurrentMessages[0].2);
   3: XIC(Message_TMR[1].EN)OTU(AOI_PlaceShip.bShipOutOfBounds);
END_ROUTINE

ROUTINE Overhead   (* ladder *)
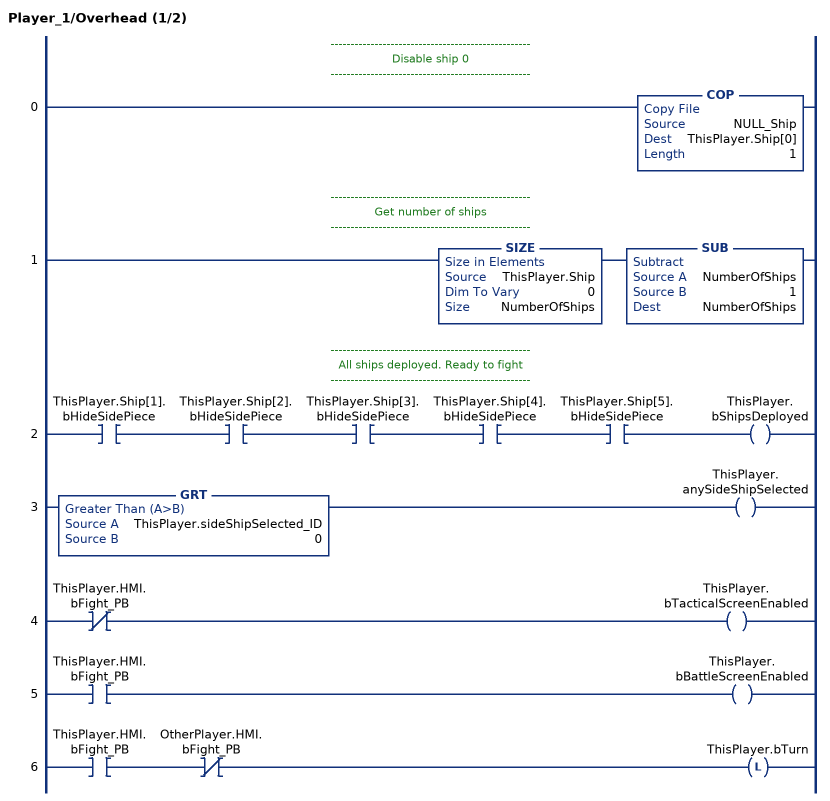
   // --------------------------------------------------
   // Disable ship 0
   // --------------------------------------------------
   0: COP(NULL_Ship,ThisPlayer.Ship[0],1);
   // --------------------------------------------------
   // Get number of ships
   // --------------------------------------------------
   1: SIZE(ThisPlayer.Ship,0,NumberOfShips)SUB(NumberOfShips,1,NumberOfShips);
   // --------------------------------------------------
   // All ships deployed. Ready to fight
   // --------------------------------------------------
   2: XIC(ThisPlayer.Ship[1].bHideSidePiece)XIC(ThisPlayer.Ship[2].bHideSidePiece)XIC(ThisPlayer.Ship[3].bHideSidePiece)XIC(ThisPlayer.Ship[4].bHideSidePiece)XIC(ThisPlayer.Ship[5].bHideSidePiece)OTE(ThisPlayer.bShipsDeployed);
   3: GRT(ThisPlayer.sideShipSelected_ID,0)OTE(ThisPlayer.anySideShipSelected);
   4: XIO(ThisPlayer.HMI.bFight_PB)OTE(ThisPlayer.bTacticalScreenEnabled);
   5: XIC(ThisPlayer.HMI.bFight_PB)OTE(ThisPlayer.bBattleScreenEnabled);
   6: XIC(ThisPlayer.HMI.bFight_PB)XIO(OtherPlayer.HMI.bFight_PB)OTL(ThisPlayer.bTurn);
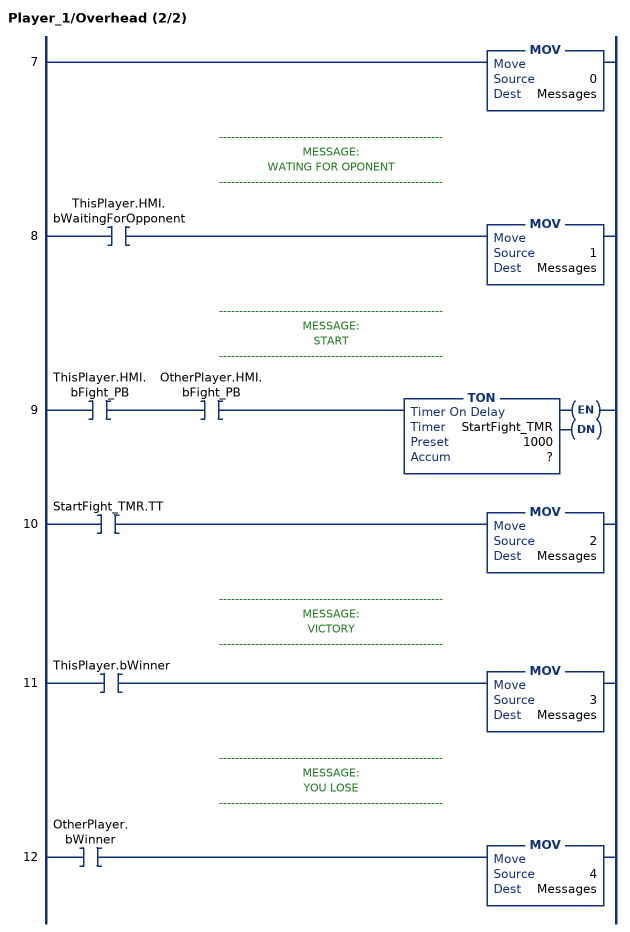
   7: MOV(0,Messages);
   // --------------------------------------------------------
   // MESSAGE:
   //   WATING FOR OPONENT
   // --------------------------------------------------------
   8: XIC(ThisPlayer.HMI.bWaitingForOpponent)MOV(1,Messages);
   // --------------------------------------------------------
   // MESSAGE:
   //   START
   // --------------------------------------------------------
   9: XIC(ThisPlayer.HMI.bFight_PB)XIC(OtherPlayer.HMI.bFight_PB)TON(StartFight_TMR,?,?);
   10: XIC(StartFight_TMR.TT)MOV(2,Messages);
   // --------------------------------------------------------
   // MESSAGE:
   //   VICTORY
   // --------------------------------------------------------
   11: XIC(ThisPlayer.bWinner)MOV(3,Messages);
   // --------------------------------------------------------
   // MESSAGE:
   //   YOU LOSE
   // --------------------------------------------------------
   12: XIC(OtherPlayer.bWinner)MOV(4,Messages);
END_ROUTINE

ROUTINE ResetBoard   (* ladder *)
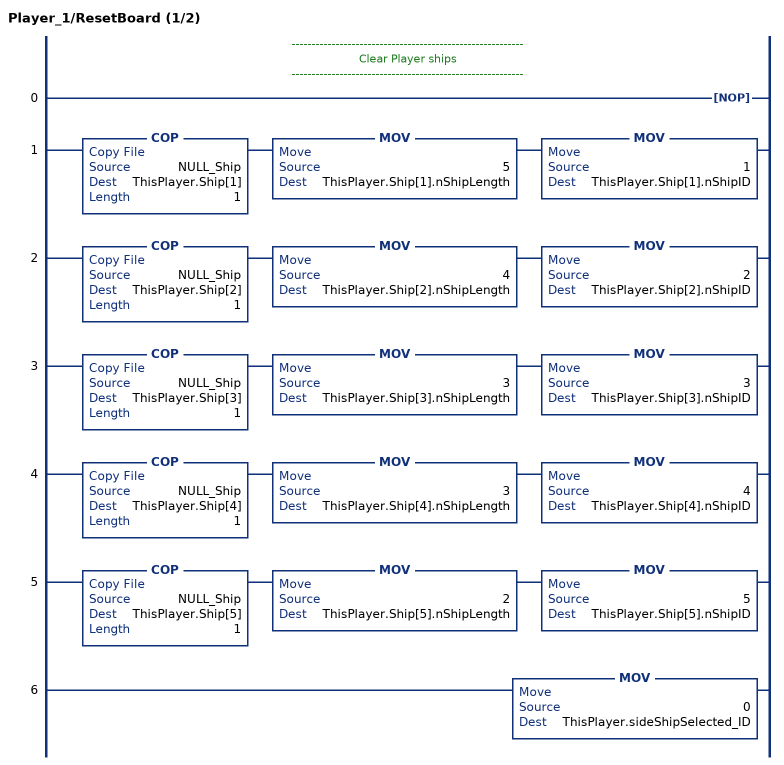
   // ----------------------------------------------------------
   // Clear Player ships
   // ----------------------------------------------------------
   0: NOP();
   1: COP(NULL_Ship,ThisPlayer.Ship[1],1)MOV(5,ThisPlayer.Ship[1].nShipLength)MOV(1,ThisPlayer.Ship[1].nShipID);
   2: COP(NULL_Ship,ThisPlayer.Ship[2],1)MOV(4,ThisPlayer.Ship[2].nShipLength)MOV(2,ThisPlayer.Ship[2].nShipID);
   3: COP(NULL_Ship,ThisPlayer.Ship[3],1)MOV(3,ThisPlayer.Ship[3].nShipLength)MOV(3,ThisPlayer.Ship[3].nShipID);
   4: COP(NULL_Ship,ThisPlayer.Ship[4],1)MOV(3,ThisPlayer.Ship[4].nShipLength)MOV(4,ThisPlayer.Ship[4].nShipID);
   5: COP(NULL_Ship,ThisPlayer.Ship[5],1)MOV(2,ThisPlayer.Ship[5].nShipLength)MOV(5,ThisPlayer.Ship[5].nShipID);
   6: MOV(0,ThisPlayer.sideShipSelected_ID);
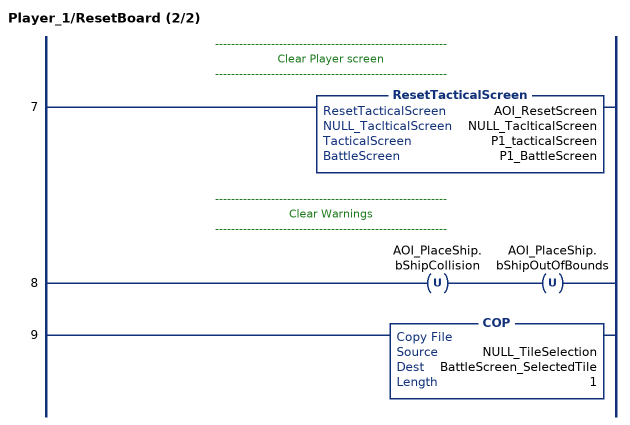
   // ----------------------------------------------------------
   // Clear Player screen
   // ----------------------------------------------------------
   7: ResetTacticalScreen(AOI_ResetScreen,NULL_TaclticalScreen,P1_tacticalScreen,P1_BattleScreen);
   // ----------------------------------------------------------
   // Clear Warnings
   // ----------------------------------------------------------
   8: OTU(AOI_PlaceShip.bShipCollision)OTU(AOI_PlaceShip.bShipOutOfBounds);
   9: COP(NULL_TileSelection,BattleScreen_SelectedTile,1);
END_ROUTINE

ROUTINE RetrieveShip   (* structured text *)
   //Initialize variables
   /*
   if not anySelected then
   	rtrv_row := -1;
   	rtrv_column := -1;
   end_if;
   */
   
   
   for rtrv_row := 0 to 9 by 1 do
   	for rtrv_column := 0 to 9 by 1 do
   		if P1_tacticalScreen[rtrv_row,rtrv_column].squareSelected AND P1_tacticalScreen[rtrv_row,rtrv_column].hasShip and not anySelected then
   
   			rtv_selectedSquare.row := rtrv_row;
   			rtv_selectedSquare.column := rtrv_column;
   			SelectedTileShipID := P1_tacticalScreen[rtrv_row,rtrv_column].ShipID;
   			anySelected := 1;
   			P1_tacticalScreen[rtrv_row,rtrv_column].squareSelected := 0;
   
   		end_if;
   	end_for;
   end_for;
   
   if anySelected then
   	for rtrv_row := 0 to 9 by 1 do
   		for rtrv_column := 0 to 9 by 1 do
   			if P1_tacticalScreen[rtrv_row,rtrv_column].ShipID = SelectedTileShipID then;
   				P1_tacticalScreen[rtrv_row,rtrv_column].IND := 2;
   
   				if P1_tacticalScreen[rtrv_row,rtrv_column].squareSelected then;
   					for rtrv_row2 := 0 to 9 by 1 do
   						for rtrv_column2 := 0 to 9 by 1 do
   							if P1_tacticalScreen[rtrv_row2,rtrv_column2].ShipID = SelectedTileShipID then;
   
   								P1_tacticalScreen[rtrv_row2,rtrv_column2].IND := 1;
   							end_if;
   						end_for;
   					end_for;
   					P1_tacticalScreen[rtrv_row,rtrv_column].squareSelected := 0;
   					anySelected := 0;
   				end_if;
   
   
   
   				if ThisPlayer.HMI.bRetrieveShip_PB then
   					//TileShipID := P1_TacticalScreen[rtrv_row,rtrv_column].hasShipType;
   					ThisPlayer.Ship[SelectedTileShipID].bHideSidePiece := 0;
   					P1_tacticalScreen[rtrv_row,rtrv_column].ShipID := -1;
   					P1_tacticalScreen[rtrv_row,rtrv_column].hasShip := 0;
   					P1_tacticalScreen[rtrv_row,rtrv_column].IND := 0;
   					anySelected := 0;
   
   
   
   				end_if;
   			end_if;
   		end_for;
   	end_for;
   end_if;
END_ROUTINE

ROUTINE SidePieces   (* structured text *)
   /*
   -------------------------------------------------------------------------------------------------------------------------------------------------------------------
   This code handles the ship pieces that get selected on the left of the tactical screen
   
   When a piece is selected (ThisPlayer.Ship[X].bIsSelected goes True), one of the one shot rising (one for every ship) gets triggered
   and the ship's ID number gets recorded in ThisPlayer.sideShipSelected_ID
   
   The counter will match the ship ID number for whichever gets triggered
   
   If a selected ship is selected again, we assign a 0 to TisPlayer.sideShipSelected_ID. This  is how we deselct a ship
   
   
   We assing a 0 to every ship that's not selected, since only one can be selected at any given time
   -------------------------------------------------------------------------------------------------------------------------------------------------------------------
   */
   
   for cntr := 1 to NumberOfShips by 1 do								// Scan from ship 1 to the last ship
   
   
   	shipSelected_OSR[cntr].InputBit := ThisPlayer.Ship[cntr].bIsSelected;
   	OSRI(shipSelected_OSR[cntr]);
   	if shipSelected_OSR[cntr].OutputBit then
   
   		if ThisPlayer.sideShipSelected_ID = 0 then
   			ThisPlayer.sideShipSelected_ID := cntr;			// Capture the ID of the piece selected
   			TacticalScreen_SelectedTile.Coordinate.row := 0;
   			TacticalScreen_SelectedTile.Coordinate.column := 0;
   
   		else
   
   
   			if ThisPlayer.sideShipSelected_ID = cntr then	// Check if the piece selected matches the one stored in memory
   
   					ThisPlayer.sideShipSelected_ID := 0;	// User deselected this ship
   
   			else
   				ThisPlayer.sideShipSelected_ID := cntr;		// Capture the ID of the piece selected
   				TacticalScreen_SelectedTile.Coordinate.row := 0;
   			TacticalScreen_SelectedTile.Coordinate.column := 0;
   
   			end_if;
   		end_if;
   
   	end_if;
   end_for;
END_ROUTINE

ROUTINE TacticalScreen   (* structured text *)
   /*
   // Initialize variables
   if not anySelected then
   	shipSelected := -1;
   	selectedSquare.row := -1;
   	selectedSquare.column := -1;
   end_if;
   
   // Look for any side ship that was selected from the side pieces
   // shipSelected = the ship the was selected from the side pieces
   for x := 0 to NumberOfShips-1 by 1  do
   	//anySelected := 0;
   	if ThisPlayer.Ship[x].isSelected then
   		shipSelected := x;
   	end_if;
   	/*
   	anySelected := ThisPlayer.Ship[x].isSelected OR anySelected;
   	if not anySelected then
   		shipSelected := -1;
   	end_if;
   
   
   end_for;
   */
   
   /*
   // If a ship piece was selected, enable search to look for the square that gets selected on the tactical screen
   // Store the XY coordinates of the selected square in selectedSquare.row and selectedSquare.column
   if ThisPlayer.sideShipSelected_ID >= 0 then
   	for row := 0 to 9 by 1 do
   		for column := 0 to 9 by 1 do
   			if P1_tacticalScreen[row,column].squareSelected then
   				selectedSquare.row := row;
   				selectedSquare.column := column;
   				P1_tacticalScreen[row,column].squareSelected := 0;
   			end_if;
   		end_for;
   	end_for;
   else
   	selectedSquare.row := -1;
   	selectedSquare.column := -1;
   end_if;
   
   // If a ship piece and a square were selected,
   // set the adjacent squares "hasShip" to 1 horizontally starting with the selected ship and moving to the left for as many squares as the ship's length
   if selectedSquare.row <> -1 AND selectedSquare.column <> -1 then
   
   	if ThisPlayer.HMI.bShipPiece_Orientation_PB then		// Place ship in vertical orientation
   		for row := selectedSquare.row to selectedSquare.row + ThisPlayer.Ship[ThisPlayer.sideShipSelected_ID].nShipLength -1 by 1 do
   			P1_tacticalScreen[row,selectedSquare.column].hasShip := 1;
   			P1_tacticalScreen[row,selectedSquare.column].ShipID := ThisPlayer.sideShipSelected_ID;
   			P1_tacticalScreen[row,selectedSquare.column].IND := 1;
   			ThisPlayer.Ship[ThisPlayer.sideShipSelected_ID].bIsSelected := 0;
   		end_for;
   
   
   	else	// Place ship in horizontal orientation
   		for column := selectedSquare.column to selectedSquare.column + ThisPlayer.Ship[ThisPlayer.sideShipSelected_ID].nShipLength -1 by 1 do
   			P1_tacticalScreen[selectedSquare.row,column].hasShip := 1;
   			P1_tacticalScreen[selectedSquare.row,column].ShipID := ThisPlayer.sideShipSelected_ID;
   			P1_tacticalScreen[selectedSquare.row,column].IND := 1;
   			ThisPlayer.Ship[ThisPlayer.sideShipSelected_ID].bIsSelected := 0;
   		end_for;
   	end_if;
   
   
   	ThisPlayer.Ship[ThisPlayer.sideShipSelected_ID].bHideSidePiece := 1;
   
   end_if;
   
   
   /*
   TODO
   
   add vertical/horizontal button and adjust how you lay the ship accordingly
   
   add retrieve button
   
   count down the ship pieces. disable piece once count reaches zero
   */
END_ROUTINE
END_PROGRAM

PROGRAM Player_2   (* main routine Main *)
VAR
   OtherPlayer : ALIAS FOR Player1;
   ThisPlayer : ALIAS FOR Player2;
END_VAR

ROUTINE CopyOtherPlayerTS   (* structured text *)
   for row := 0 to 10 by 1 do
   	for column := 0 to 10 by 1 do
   		cop(P1_tacticalScreen[row,column], P2_tacticalScreen[row,column], 1);
   	end_for;
   end_for;
END_ROUTINE

ROUTINE Main   (* ladder *)
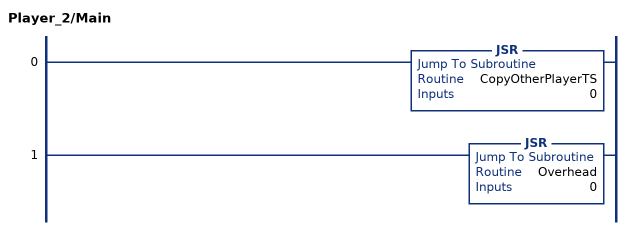
   0: JSR(CopyOtherPlayerTS,0);
   1: JSR(Overhead,0);
END_ROUTINE

ROUTINE Overhead   (* ladder *)
END_ROUTINE
END_PROGRAM
